(* IEC 61131-3 sources: Lasal/CPU_5344_V01/Class/Bit2ByteConversion_outputs, 1 file *)

(* ---- Bit2ByteConversion_outputs.st ---- *)
(*!
<Class
	Name               = "Bit2ByteConversion_outputs"
	Revision           = "0.1"
	RealtimeTask       = "false"
	CyclicTask         = "false"
	BackgroundTask     = "false"
	Sigmatek           = "false"
	OSInterface        = "false"
	HighPriority       = "false"
	Automatic          = "false"
	UpdateMode         = "Prescan"
	SharedCommandTable = "true"
	Objectsize         = "(390,2040)">
	<Channels>
		<Server Name="Bit1" Visualized="true" Initialize="false" WriteProtected="false" Retentive="false"/>
		<Server Name="Bit10" Visualized="true" Initialize="false" WriteProtected="false" Retentive="false"/>
		<Server Name="Bit11" Visualized="true" Initialize="false" WriteProtected="false" Retentive="false"/>
		<Server Name="Bit12" Visualized="true" Initialize="false" WriteProtected="false" Retentive="false"/>
		<Server Name="Bit13" Visualized="true" Initialize="false" WriteProtected="false" Retentive="false"/>
		<Server Name="Bit14" Visualized="true" Initialize="false" WriteProtected="false" Retentive="false"/>
		<Server Name="Bit15" Visualized="true" Initialize="false" WriteProtected="false" Retentive="false"/>
		<Server Name="Bit16" Visualized="true" Initialize="false" WriteProtected="false" Retentive="false"/>
		<Server Name="Bit17" Visualized="true" Initialize="false" WriteProtected="false" Retentive="false"/>
		<Server Name="Bit18" Visualized="true" Initialize="false" WriteProtected="false" Retentive="false"/>
		<Server Name="Bit19" Visualized="true" Initialize="false" WriteProtected="false" Retentive="false"/>
		<Server Name="Bit2" Visualized="true" Initialize="false" WriteProtected="false" Retentive="false"/>
		<Server Name="Bit20" Visualized="true" Initialize="false" WriteProtected="false" Retentive="false"/>
		<Server Name="Bit21" Visualized="true" Initialize="false" WriteProtected="false" Retentive="false"/>
		<Server Name="Bit22" Visualized="true" Initialize="false" WriteProtected="false" Retentive="false"/>
		<Server Name="Bit23" Visualized="true" Initialize="false" WriteProtected="false" Retentive="false"/>
		<Server Name="Bit24" Visualized="true" Initialize="false" WriteProtected="false" Retentive="false"/>
		<Server Name="Bit25" Visualized="true" Initialize="false" WriteProtected="false" Retentive="false"/>
		<Server Name="Bit26" Visualized="true" Initialize="false" WriteProtected="false" Retentive="false"/>
		<Server Name="Bit27" Visualized="true" Initialize="false" WriteProtected="false" Retentive="false"/>
		<Server Name="Bit28" Visualized="true" Initialize="false" WriteProtected="false" Retentive="false"/>
		<Server Name="Bit29" Visualized="true" Initialize="false" WriteProtected="false" Retentive="false"/>
		<Server Name="Bit3" Visualized="true" Initialize="false" WriteProtected="false" Retentive="false"/>
		<Server Name="Bit30" Visualized="true" Initialize="false" WriteProtected="false" Retentive="false"/>
		<Server Name="Bit31" Visualized="true" Initialize="false" WriteProtected="false" Retentive="false"/>
		<Server Name="Bit32" Visualized="true" Initialize="false" WriteProtected="false" Retentive="false"/>
		<Server Name="Bit4" Visualized="true" Initialize="false" WriteProtected="false" Retentive="false"/>
		<Server Name="Bit5" Visualized="true" Initialize="false" WriteProtected="false" Retentive="false"/>
		<Server Name="Bit6" Visualized="true" Initialize="false" WriteProtected="false" Retentive="false"/>
		<Server Name="Bit7" Visualized="true" Initialize="false" WriteProtected="false" Retentive="false"/>
		<Server Name="Bit8" Visualized="true" Initialize="false" WriteProtected="false" Retentive="false"/>
		<Server Name="Bit9" Visualized="true" Initialize="false" WriteProtected="false" Retentive="false"/>
		<Server Name="BitValue" Visualized="false" Initialize="false" WriteProtected="true" Retentive="false"/>
		<Client Name="BValue" Required="false" Internal="false"/>
	</Channels>
	<RevDoku>
		<Owner Company="Intecon" Author="Richard Fierkens"/>
		<Dokumentation Revision="0.1" Date="2011-12-28" Author="Richard Fierkens" Company="Intecon" Description="Write timedelay is removed.&#13;&#10;Read timedelay is set to 10mSec."/>
		<Dokumentation Revision="0.0" Date="2011-12-27" Author="Johan Embregts" Company="SigmaControl" Description="Created."/>
	</RevDoku>
</Class>
*)
Bit2ByteConversion_outputs : CLASS
  //Servers:
	BitValue 	: SvrChCmd_BDINT;
	Bit1 	: SvrCh_DINT;
	Bit2 	: SvrCh_DINT;
	Bit3 	: SvrCh_DINT;
	Bit4 	: SvrCh_DINT;
	Bit5 	: SvrCh_DINT;
	Bit6 	: SvrCh_DINT;
	Bit7 	: SvrCh_DINT;
	Bit8 	: SvrCh_DINT;
	Bit9 	: SvrCh_DINT;
	Bit10 	: SvrCh_DINT;
	Bit11 	: SvrCh_DINT;
	Bit12 	: SvrCh_DINT;
	Bit13 	: SvrCh_DINT;
	Bit14 	: SvrCh_DINT;
	Bit15 	: SvrCh_DINT;
	Bit16 	: SvrCh_DINT;
	Bit17 	: SvrCh_DINT;
	Bit18 	: SvrCh_DINT;
	Bit19 	: SvrCh_DINT;
	Bit20 	: SvrCh_DINT;
	Bit21 	: SvrCh_DINT;
	Bit22 	: SvrCh_DINT;
	Bit23 	: SvrCh_DINT;
	Bit24 	: SvrCh_DINT;
	Bit25 	: SvrCh_DINT;
	Bit26 	: SvrCh_DINT;
	Bit27 	: SvrCh_DINT;
	Bit28 	: SvrCh_DINT;
	Bit29 	: SvrCh_DINT;
	Bit30 	: SvrCh_DINT;
	Bit31 	: SvrCh_DINT;
	Bit32 	: SvrCh_DINT;
  //Clients:
	BValue 	: CltCh_BDINT;
  //Variables:
		tMark 	: UDINT;
  //Functions:

	FUNCTION VIRTUAL ReadMe;

	FUNCTION VIRTUAL WriteMe;

	FUNCTION VIRTUAL GLOBAL Bit1::Read
		VAR_OUTPUT
			output (EAX) 	: DINT;
		END_VAR;

	FUNCTION VIRTUAL GLOBAL Bit1::Write
		VAR_INPUT
			input (EAX) 	: DINT;
		END_VAR
		VAR_OUTPUT
			result (EAX) 	: DINT;
		END_VAR;

	FUNCTION VIRTUAL GLOBAL Bit2::Read
		VAR_OUTPUT
			output (EAX) 	: DINT;
		END_VAR;

	FUNCTION VIRTUAL GLOBAL Bit2::Write
		VAR_INPUT
			input (EAX) 	: DINT;
		END_VAR
		VAR_OUTPUT
			result (EAX) 	: DINT;
		END_VAR;

	FUNCTION VIRTUAL GLOBAL Bit3::Read
		VAR_OUTPUT
			output (EAX) 	: DINT;
		END_VAR;

	FUNCTION VIRTUAL GLOBAL Bit3::Write
		VAR_INPUT
			input (EAX) 	: DINT;
		END_VAR
		VAR_OUTPUT
			result (EAX) 	: DINT;
		END_VAR;

	FUNCTION VIRTUAL GLOBAL Bit4::Read
		VAR_OUTPUT
			output (EAX) 	: DINT;
		END_VAR;

	FUNCTION VIRTUAL GLOBAL Bit4::Write
		VAR_INPUT
			input (EAX) 	: DINT;
		END_VAR
		VAR_OUTPUT
			result (EAX) 	: DINT;
		END_VAR;

	FUNCTION VIRTUAL GLOBAL Bit5::Read
		VAR_OUTPUT
			output (EAX) 	: DINT;
		END_VAR;

	FUNCTION VIRTUAL GLOBAL Bit5::Write
		VAR_INPUT
			input (EAX) 	: DINT;
		END_VAR
		VAR_OUTPUT
			result (EAX) 	: DINT;
		END_VAR;

	FUNCTION VIRTUAL GLOBAL Bit6::Read
		VAR_OUTPUT
			output (EAX) 	: DINT;
		END_VAR;

	FUNCTION VIRTUAL GLOBAL Bit6::Write
		VAR_INPUT
			input (EAX) 	: DINT;
		END_VAR
		VAR_OUTPUT
			result (EAX) 	: DINT;
		END_VAR;

	FUNCTION VIRTUAL GLOBAL Bit7::Read
		VAR_OUTPUT
			output (EAX) 	: DINT;
		END_VAR;

	FUNCTION VIRTUAL GLOBAL Bit7::Write
		VAR_INPUT
			input (EAX) 	: DINT;
		END_VAR
		VAR_OUTPUT
			result (EAX) 	: DINT;
		END_VAR;

	FUNCTION VIRTUAL GLOBAL Bit8::Read
		VAR_OUTPUT
			output (EAX) 	: DINT;
		END_VAR;

	FUNCTION VIRTUAL GLOBAL Bit8::Write
		VAR_INPUT
			input (EAX) 	: DINT;
		END_VAR
		VAR_OUTPUT
			result (EAX) 	: DINT;
		END_VAR;

	FUNCTION VIRTUAL GLOBAL Bit9::Read
		VAR_OUTPUT
			output (EAX) 	: DINT;
		END_VAR;

	FUNCTION VIRTUAL GLOBAL Bit9::Write
		VAR_INPUT
			input (EAX) 	: DINT;
		END_VAR
		VAR_OUTPUT
			result (EAX) 	: DINT;
		END_VAR;

	FUNCTION VIRTUAL GLOBAL Bit10::Read
		VAR_OUTPUT
			output (EAX) 	: DINT;
		END_VAR;

	FUNCTION VIRTUAL GLOBAL Bit10::Write
		VAR_INPUT
			input (EAX) 	: DINT;
		END_VAR
		VAR_OUTPUT
			result (EAX) 	: DINT;
		END_VAR;

	FUNCTION VIRTUAL GLOBAL Bit11::Read
		VAR_OUTPUT
			output (EAX) 	: DINT;
		END_VAR;

	FUNCTION VIRTUAL GLOBAL Bit11::Write
		VAR_INPUT
			input (EAX) 	: DINT;
		END_VAR
		VAR_OUTPUT
			result (EAX) 	: DINT;
		END_VAR;

	FUNCTION VIRTUAL GLOBAL Bit12::Read
		VAR_OUTPUT
			output (EAX) 	: DINT;
		END_VAR;

	FUNCTION VIRTUAL GLOBAL Bit12::Write
		VAR_INPUT
			input (EAX) 	: DINT;
		END_VAR
		VAR_OUTPUT
			result (EAX) 	: DINT;
		END_VAR;

	FUNCTION VIRTUAL GLOBAL Bit13::Read
		VAR_OUTPUT
			output (EAX) 	: DINT;
		END_VAR;

	FUNCTION VIRTUAL GLOBAL Bit13::Write
		VAR_INPUT
			input (EAX) 	: DINT;
		END_VAR
		VAR_OUTPUT
			result (EAX) 	: DINT;
		END_VAR;

	FUNCTION VIRTUAL GLOBAL Bit14::Read
		VAR_OUTPUT
			output (EAX) 	: DINT;
		END_VAR;

	FUNCTION VIRTUAL GLOBAL Bit14::Write
		VAR_INPUT
			input (EAX) 	: DINT;
		END_VAR
		VAR_OUTPUT
			result (EAX) 	: DINT;
		END_VAR;

	FUNCTION VIRTUAL GLOBAL Bit15::Read
		VAR_OUTPUT
			output (EAX) 	: DINT;
		END_VAR;

	FUNCTION VIRTUAL GLOBAL Bit15::Write
		VAR_INPUT
			input (EAX) 	: DINT;
		END_VAR
		VAR_OUTPUT
			result (EAX) 	: DINT;
		END_VAR;

	FUNCTION VIRTUAL GLOBAL Bit16::Read
		VAR_OUTPUT
			output (EAX) 	: DINT;
		END_VAR;

	FUNCTION VIRTUAL GLOBAL Bit16::Write
		VAR_INPUT
			input (EAX) 	: DINT;
		END_VAR
		VAR_OUTPUT
			result (EAX) 	: DINT;
		END_VAR;

	FUNCTION VIRTUAL GLOBAL Bit17::Read
		VAR_OUTPUT
			output (EAX) 	: DINT;
		END_VAR;

	FUNCTION VIRTUAL GLOBAL Bit17::Write
		VAR_INPUT
			input (EAX) 	: DINT;
		END_VAR
		VAR_OUTPUT
			result (EAX) 	: DINT;
		END_VAR;

	FUNCTION VIRTUAL GLOBAL Bit18::Read
		VAR_OUTPUT
			output (EAX) 	: DINT;
		END_VAR;

	FUNCTION VIRTUAL GLOBAL Bit18::Write
		VAR_INPUT
			input (EAX) 	: DINT;
		END_VAR
		VAR_OUTPUT
			result (EAX) 	: DINT;
		END_VAR;

	FUNCTION VIRTUAL GLOBAL Bit19::Read
		VAR_OUTPUT
			output (EAX) 	: DINT;
		END_VAR;

	FUNCTION VIRTUAL GLOBAL Bit19::Write
		VAR_INPUT
			input (EAX) 	: DINT;
		END_VAR
		VAR_OUTPUT
			result (EAX) 	: DINT;
		END_VAR;

	FUNCTION VIRTUAL GLOBAL Bit20::Read
		VAR_OUTPUT
			output (EAX) 	: DINT;
		END_VAR;

	FUNCTION VIRTUAL GLOBAL Bit20::Write
		VAR_INPUT
			input (EAX) 	: DINT;
		END_VAR
		VAR_OUTPUT
			result (EAX) 	: DINT;
		END_VAR;

	FUNCTION VIRTUAL GLOBAL Bit21::Read
		VAR_OUTPUT
			output (EAX) 	: DINT;
		END_VAR;

	FUNCTION VIRTUAL GLOBAL Bit21::Write
		VAR_INPUT
			input (EAX) 	: DINT;
		END_VAR
		VAR_OUTPUT
			result (EAX) 	: DINT;
		END_VAR;

	FUNCTION VIRTUAL GLOBAL Bit22::Read
		VAR_OUTPUT
			output (EAX) 	: DINT;
		END_VAR;

	FUNCTION VIRTUAL GLOBAL Bit22::Write
		VAR_INPUT
			input (EAX) 	: DINT;
		END_VAR
		VAR_OUTPUT
			result (EAX) 	: DINT;
		END_VAR;

	FUNCTION VIRTUAL GLOBAL Bit23::Read
		VAR_OUTPUT
			output (EAX) 	: DINT;
		END_VAR;

	FUNCTION VIRTUAL GLOBAL Bit23::Write
		VAR_INPUT
			input (EAX) 	: DINT;
		END_VAR
		VAR_OUTPUT
			result (EAX) 	: DINT;
		END_VAR;

	FUNCTION VIRTUAL GLOBAL Bit24::Read
		VAR_OUTPUT
			output (EAX) 	: DINT;
		END_VAR;

	FUNCTION VIRTUAL GLOBAL Bit24::Write
		VAR_INPUT
			input (EAX) 	: DINT;
		END_VAR
		VAR_OUTPUT
			result (EAX) 	: DINT;
		END_VAR;

	FUNCTION VIRTUAL GLOBAL Bit25::Read
		VAR_OUTPUT
			output (EAX) 	: DINT;
		END_VAR;

	FUNCTION VIRTUAL GLOBAL Bit25::Write
		VAR_INPUT
			input (EAX) 	: DINT;
		END_VAR
		VAR_OUTPUT
			result (EAX) 	: DINT;
		END_VAR;

	FUNCTION VIRTUAL GLOBAL Bit26::Read
		VAR_OUTPUT
			output (EAX) 	: DINT;
		END_VAR;

	FUNCTION VIRTUAL GLOBAL Bit26::Write
		VAR_INPUT
			input (EAX) 	: DINT;
		END_VAR
		VAR_OUTPUT
			result (EAX) 	: DINT;
		END_VAR;

	FUNCTION VIRTUAL GLOBAL Bit27::Read
		VAR_OUTPUT
			output (EAX) 	: DINT;
		END_VAR;

	FUNCTION VIRTUAL GLOBAL Bit27::Write
		VAR_INPUT
			input (EAX) 	: DINT;
		END_VAR
		VAR_OUTPUT
			result (EAX) 	: DINT;
		END_VAR;

	FUNCTION VIRTUAL GLOBAL Bit28::Read
		VAR_OUTPUT
			output (EAX) 	: DINT;
		END_VAR;

	FUNCTION VIRTUAL GLOBAL Bit28::Write
		VAR_INPUT
			input (EAX) 	: DINT;
		END_VAR
		VAR_OUTPUT
			result (EAX) 	: DINT;
		END_VAR;

	FUNCTION VIRTUAL GLOBAL Bit29::Read
		VAR_OUTPUT
			output (EAX) 	: DINT;
		END_VAR;

	FUNCTION VIRTUAL GLOBAL Bit29::Write
		VAR_INPUT
			input (EAX) 	: DINT;
		END_VAR
		VAR_OUTPUT
			result (EAX) 	: DINT;
		END_VAR;

	FUNCTION VIRTUAL GLOBAL Bit30::Read
		VAR_OUTPUT
			output (EAX) 	: DINT;
		END_VAR;

	FUNCTION VIRTUAL GLOBAL Bit30::Write
		VAR_INPUT
			input (EAX) 	: DINT;
		END_VAR
		VAR_OUTPUT
			result (EAX) 	: DINT;
		END_VAR;

	FUNCTION VIRTUAL GLOBAL Bit31::Read
		VAR_OUTPUT
			output (EAX) 	: DINT;
		END_VAR;

	FUNCTION VIRTUAL GLOBAL Bit31::Write
		VAR_INPUT
			input (EAX) 	: DINT;
		END_VAR
		VAR_OUTPUT
			result (EAX) 	: DINT;
		END_VAR;

	FUNCTION VIRTUAL GLOBAL Bit32::Read
		VAR_OUTPUT
			output (EAX) 	: DINT;
		END_VAR;

	FUNCTION VIRTUAL GLOBAL Bit32::Write
		VAR_INPUT
			input (EAX) 	: DINT;
		END_VAR
		VAR_OUTPUT
			result (EAX) 	: DINT;
		END_VAR;
  //Tables:
	FUNCTION @STD
		VAR_OUTPUT
			ret_code	: CONFSTATES;
		END_VAR;
	FUNCTION GLOBAL TAB @CT_;
END_CLASS;

#define cMaxUpdateTime  10 // mSec

FUNCTION VIRTUAL GLOBAL Bit2ByteConversion_outputs::Bit1::Read
	VAR_OUTPUT
		output (EAX) 	: DINT;
	END_VAR

  ReadMe();
	output := Bit1;

END_FUNCTION

FUNCTION VIRTUAL GLOBAL Bit2ByteConversion_outputs::Bit2::Read
	VAR_OUTPUT
		output (EAX) 	: DINT;
	END_VAR

  ReadMe();
	output := Bit2;

END_FUNCTION

FUNCTION VIRTUAL GLOBAL Bit2ByteConversion_outputs::Bit3::Read
	VAR_OUTPUT
		output (EAX) 	: DINT;
	END_VAR

  ReadMe();
	output := Bit3;

END_FUNCTION

FUNCTION VIRTUAL GLOBAL Bit2ByteConversion_outputs::Bit4::Read
	VAR_OUTPUT
		output (EAX) 	: DINT;
	END_VAR

  ReadMe();
	output := Bit4;

END_FUNCTION

FUNCTION VIRTUAL GLOBAL Bit2ByteConversion_outputs::Bit5::Read
	VAR_OUTPUT
		output (EAX) 	: DINT;
	END_VAR

  ReadMe();
	output := Bit5;

END_FUNCTION

FUNCTION VIRTUAL GLOBAL Bit2ByteConversion_outputs::Bit6::Read
	VAR_OUTPUT
		output (EAX) 	: DINT;
	END_VAR

  ReadMe();
	output := Bit6;

END_FUNCTION

FUNCTION VIRTUAL GLOBAL Bit2ByteConversion_outputs::Bit7::Read
	VAR_OUTPUT
		output (EAX) 	: DINT;
	END_VAR

  ReadMe();
	output := Bit7;

END_FUNCTION

FUNCTION VIRTUAL GLOBAL Bit2ByteConversion_outputs::Bit8::Read
	VAR_OUTPUT
		output (EAX) 	: DINT;
	END_VAR

  ReadMe();
	output := Bit8;

END_FUNCTION

FUNCTION VIRTUAL GLOBAL Bit2ByteConversion_outputs::Bit9::Read
	VAR_OUTPUT
		output (EAX) 	: DINT;
	END_VAR

  ReadMe();
	output := Bit9;

END_FUNCTION

FUNCTION VIRTUAL GLOBAL Bit2ByteConversion_outputs::Bit10::Read
	VAR_OUTPUT
		output (EAX) 	: DINT;
	END_VAR

  ReadMe();
	output := Bit10;

END_FUNCTION

FUNCTION VIRTUAL GLOBAL Bit2ByteConversion_outputs::Bit11::Read
	VAR_OUTPUT
		output (EAX) 	: DINT;
	END_VAR

  ReadMe();
	output := Bit11;

END_FUNCTION

FUNCTION VIRTUAL GLOBAL Bit2ByteConversion_outputs::Bit12::Read
	VAR_OUTPUT
		output (EAX) 	: DINT;
	END_VAR

  ReadMe();
	output := Bit12;

END_FUNCTION

FUNCTION VIRTUAL GLOBAL Bit2ByteConversion_outputs::Bit13::Read
	VAR_OUTPUT
		output (EAX) 	: DINT;
	END_VAR

  ReadMe();
	output := Bit13;

END_FUNCTION

FUNCTION VIRTUAL GLOBAL Bit2ByteConversion_outputs::Bit14::Read
	VAR_OUTPUT
		output (EAX) 	: DINT;
	END_VAR

  ReadMe();
	output := Bit14;

END_FUNCTION

FUNCTION VIRTUAL GLOBAL Bit2ByteConversion_outputs::Bit15::Read
	VAR_OUTPUT
		output (EAX) 	: DINT;
	END_VAR

  ReadMe();
	output := Bit15;

END_FUNCTION

FUNCTION VIRTUAL GLOBAL Bit2ByteConversion_outputs::Bit16::Read
	VAR_OUTPUT
		output (EAX) 	: DINT;
	END_VAR

  ReadMe();
	output := Bit16;

END_FUNCTION

FUNCTION VIRTUAL GLOBAL Bit2ByteConversion_outputs::Bit17::Read
	VAR_OUTPUT
		output (EAX) 	: DINT;
	END_VAR

  ReadMe();
	output := Bit17;

END_FUNCTION

FUNCTION VIRTUAL GLOBAL Bit2ByteConversion_outputs::Bit18::Read
	VAR_OUTPUT
		output (EAX) 	: DINT;
	END_VAR

  ReadMe();
	output := Bit18;

END_FUNCTION

FUNCTION VIRTUAL GLOBAL Bit2ByteConversion_outputs::Bit19::Read
	VAR_OUTPUT
		output (EAX) 	: DINT;
	END_VAR

  ReadMe();
	output := Bit19;

END_FUNCTION

FUNCTION VIRTUAL GLOBAL Bit2ByteConversion_outputs::Bit20::Read
	VAR_OUTPUT
		output (EAX) 	: DINT;
	END_VAR

  ReadMe();
	output := Bit20;

END_FUNCTION

FUNCTION VIRTUAL GLOBAL Bit2ByteConversion_outputs::Bit21::Read
	VAR_OUTPUT
		output (EAX) 	: DINT;
	END_VAR

  ReadMe();
	output := Bit21;

END_FUNCTION

FUNCTION VIRTUAL GLOBAL Bit2ByteConversion_outputs::Bit22::Read
	VAR_OUTPUT
		output (EAX) 	: DINT;
	END_VAR

  ReadMe();
	output := Bit22;

END_FUNCTION

FUNCTION VIRTUAL GLOBAL Bit2ByteConversion_outputs::Bit23::Read
	VAR_OUTPUT
		output (EAX) 	: DINT;
	END_VAR

  ReadMe();
	output := Bit23;

END_FUNCTION

FUNCTION VIRTUAL GLOBAL Bit2ByteConversion_outputs::Bit24::Read
	VAR_OUTPUT
		output (EAX) 	: DINT;
	END_VAR

  ReadMe();
	output := Bit24;

END_FUNCTION

FUNCTION VIRTUAL GLOBAL Bit2ByteConversion_outputs::Bit25::Read
	VAR_OUTPUT
		output (EAX) 	: DINT;
	END_VAR

  ReadMe();
	output := Bit25;

END_FUNCTION

FUNCTION VIRTUAL GLOBAL Bit2ByteConversion_outputs::Bit26::Read
	VAR_OUTPUT
		output (EAX) 	: DINT;
	END_VAR

  ReadMe();
	output := Bit26;

END_FUNCTION

FUNCTION VIRTUAL GLOBAL Bit2ByteConversion_outputs::Bit27::Read
	VAR_OUTPUT
		output (EAX) 	: DINT;
	END_VAR

  ReadMe();
	output := Bit27;

END_FUNCTION

FUNCTION VIRTUAL GLOBAL Bit2ByteConversion_outputs::Bit28::Read
	VAR_OUTPUT
		output (EAX) 	: DINT;
	END_VAR

  ReadMe();
	output := Bit28;

END_FUNCTION

FUNCTION VIRTUAL GLOBAL Bit2ByteConversion_outputs::Bit29::Read
	VAR_OUTPUT
		output (EAX) 	: DINT;
	END_VAR

  ReadMe();
	output := Bit29;

END_FUNCTION

FUNCTION VIRTUAL GLOBAL Bit2ByteConversion_outputs::Bit30::Read
	VAR_OUTPUT
		output (EAX) 	: DINT;
	END_VAR

  ReadMe();
	output := Bit30;

END_FUNCTION

FUNCTION VIRTUAL GLOBAL Bit2ByteConversion_outputs::Bit31::Read
	VAR_OUTPUT
		output (EAX) 	: DINT;
	END_VAR

  ReadMe();
	output := Bit31;

END_FUNCTION

FUNCTION VIRTUAL GLOBAL Bit2ByteConversion_outputs::Bit32::Read
	VAR_OUTPUT
		output (EAX) 	: DINT;
	END_VAR

  ReadMe();
	output := Bit32;

END_FUNCTION

FUNCTION VIRTUAL GLOBAL Bit2ByteConversion_outputs::Bit1::Write
	VAR_INPUT
		input (EAX) 	: DINT;
	END_VAR
	VAR_OUTPUT
		result (EAX) 	: DINT;
	END_VAR

  Bit1 := input and 2#1;
	BValue.1 := to_Bool( Bit1);
  WriteMe();
 	result := Bit1;

END_FUNCTION

FUNCTION VIRTUAL GLOBAL Bit2ByteConversion_outputs::Bit2::Write
	VAR_INPUT
		input (EAX) 	: DINT;
	END_VAR
	VAR_OUTPUT
		result (EAX) 	: DINT;
	END_VAR

  Bit2 := input and 2#1;
	BValue.2 := to_Bool( Bit2);
  WriteMe();
 	result := Bit2;

END_FUNCTION

FUNCTION VIRTUAL GLOBAL Bit2ByteConversion_outputs::Bit3::Write
	VAR_INPUT
		input (EAX) 	: DINT;
	END_VAR
	VAR_OUTPUT
		result (EAX) 	: DINT;
	END_VAR

  Bit3 := input and 2#1;
	BValue.3 := to_Bool( Bit3);
  WriteMe();
 	result := Bit3;

END_FUNCTION

FUNCTION VIRTUAL GLOBAL Bit2ByteConversion_outputs::Bit4::Write
	VAR_INPUT
		input (EAX) 	: DINT;
	END_VAR
	VAR_OUTPUT
		result (EAX) 	: DINT;
	END_VAR

  Bit4 := input and 2#1;
	BValue.4 := to_Bool( Bit4);
  WriteMe();
 	result := Bit4;

END_FUNCTION

FUNCTION VIRTUAL GLOBAL Bit2ByteConversion_outputs::Bit5::Write
	VAR_INPUT
		input (EAX) 	: DINT;
	END_VAR
	VAR_OUTPUT
		result (EAX) 	: DINT;
	END_VAR

  Bit5 := input and 2#1;
	BValue.5 := to_Bool( Bit5);
  WriteMe();
 	result := Bit5;

END_FUNCTION

FUNCTION VIRTUAL GLOBAL Bit2ByteConversion_outputs::Bit6::Write
	VAR_INPUT
		input (EAX) 	: DINT;
	END_VAR
	VAR_OUTPUT
		result (EAX) 	: DINT;
	END_VAR

  Bit6 := input and 2#1;
	BValue.6 := to_Bool( Bit6);
  WriteMe();
 	result := Bit6;

END_FUNCTION

FUNCTION VIRTUAL GLOBAL Bit2ByteConversion_outputs::Bit7::Write
	VAR_INPUT
		input (EAX) 	: DINT;
	END_VAR
	VAR_OUTPUT
		result (EAX) 	: DINT;
	END_VAR

  Bit7 := input and 2#1;
	BValue.7 := to_Bool( Bit7);
  WriteMe();
 	result := Bit7;

END_FUNCTION

FUNCTION VIRTUAL GLOBAL Bit2ByteConversion_outputs::Bit8::Write
	VAR_INPUT
		input (EAX) 	: DINT;
	END_VAR
	VAR_OUTPUT
		result (EAX) 	: DINT;
	END_VAR

  Bit8 := input and 2#1;
	BValue.8 := to_Bool( Bit8);
  WriteMe();
 	result := Bit8;

END_FUNCTION

FUNCTION VIRTUAL GLOBAL Bit2ByteConversion_outputs::Bit9::Write
	VAR_INPUT
		input (EAX) 	: DINT;
	END_VAR
	VAR_OUTPUT
		result (EAX) 	: DINT;
	END_VAR

  Bit9 := input and 2#1;
	BValue.9 := to_Bool( Bit9);
  WriteMe();
 	result := Bit9;

END_FUNCTION

FUNCTION VIRTUAL GLOBAL Bit2ByteConversion_outputs::Bit10::Write
	VAR_INPUT
		input (EAX) 	: DINT;
	END_VAR
	VAR_OUTPUT
		result (EAX) 	: DINT;
	END_VAR

  Bit10 := input and 2#1;
	BValue.10 := to_Bool( Bit10);
  WriteMe();
 	result := Bit10;

END_FUNCTION

FUNCTION VIRTUAL GLOBAL Bit2ByteConversion_outputs::Bit11::Write
	VAR_INPUT
		input (EAX) 	: DINT;
	END_VAR
	VAR_OUTPUT
		result (EAX) 	: DINT;
	END_VAR

  Bit11 := input and 2#1;
	BValue.11 := to_Bool( Bit11);
  WriteMe();
 	result := Bit11;

END_FUNCTION

FUNCTION VIRTUAL GLOBAL Bit2ByteConversion_outputs::Bit12::Write
	VAR_INPUT
		input (EAX) 	: DINT;
	END_VAR
	VAR_OUTPUT
		result (EAX) 	: DINT;
	END_VAR

  Bit12 := input and 2#1;
	BValue.12 := to_Bool( Bit12);
  WriteMe();
 	result := Bit12;

END_FUNCTION

FUNCTION VIRTUAL GLOBAL Bit2ByteConversion_outputs::Bit13::Write
	VAR_INPUT
		input (EAX) 	: DINT;
	END_VAR
	VAR_OUTPUT
		result (EAX) 	: DINT;
	END_VAR

  Bit13 := input and 2#1;
	BValue.13 := to_Bool( Bit13);
  WriteMe();
 	result := Bit13;

END_FUNCTION

FUNCTION VIRTUAL GLOBAL Bit2ByteConversion_outputs::Bit14::Write
	VAR_INPUT
		input (EAX) 	: DINT;
	END_VAR
	VAR_OUTPUT
		result (EAX) 	: DINT;
	END_VAR

  Bit14 := input and 2#1;
	BValue.14 := to_Bool( Bit14);
  WriteMe();
 	result := Bit14;

END_FUNCTION

FUNCTION VIRTUAL GLOBAL Bit2ByteConversion_outputs::Bit15::Write
	VAR_INPUT
		input (EAX) 	: DINT;
	END_VAR
	VAR_OUTPUT
		result (EAX) 	: DINT;
	END_VAR

  Bit15 := input and 2#1;
	BValue.15 := to_Bool( Bit15);
  WriteMe();
 	result := Bit15;

END_FUNCTION

FUNCTION VIRTUAL GLOBAL Bit2ByteConversion_outputs::Bit16::Write
	VAR_INPUT
		input (EAX) 	: DINT;
	END_VAR
	VAR_OUTPUT
		result (EAX) 	: DINT;
	END_VAR

  Bit16 := input and 2#1;
	BValue.16 := to_Bool( Bit16);
  WriteMe();
 	result := Bit16;

END_FUNCTION

FUNCTION VIRTUAL GLOBAL Bit2ByteConversion_outputs::Bit17::Write
	VAR_INPUT
		input (EAX) 	: DINT;
	END_VAR
	VAR_OUTPUT
		result (EAX) 	: DINT;
	END_VAR

  Bit17 := input and 2#1;
	BValue.17 := to_Bool( Bit17);
  WriteMe();
 	result := Bit17;

END_FUNCTION

FUNCTION VIRTUAL GLOBAL Bit2ByteConversion_outputs::Bit18::Write
	VAR_INPUT
		input (EAX) 	: DINT;
	END_VAR
	VAR_OUTPUT
		result (EAX) 	: DINT;
	END_VAR

  Bit18 := input and 2#1;
	BValue.18 := to_Bool( Bit18);
  WriteMe();
 	result := Bit18;

END_FUNCTION

FUNCTION VIRTUAL GLOBAL Bit2ByteConversion_outputs::Bit19::Write
	VAR_INPUT
		input (EAX) 	: DINT;
	END_VAR
	VAR_OUTPUT
		result (EAX) 	: DINT;
	END_VAR

  Bit19 := input and 2#1;
	BValue.19 := to_Bool( Bit19);
  WriteMe();
 	result := Bit19;

END_FUNCTION

FUNCTION VIRTUAL GLOBAL Bit2ByteConversion_outputs::Bit20::Write
	VAR_INPUT
		input (EAX) 	: DINT;
	END_VAR
	VAR_OUTPUT
		result (EAX) 	: DINT;
	END_VAR

  Bit20 := input and 2#1;
	BValue.20 := to_Bool( Bit20);
  WriteMe();
 	result := Bit20;

END_FUNCTION

FUNCTION VIRTUAL GLOBAL Bit2ByteConversion_outputs::Bit21::Write
	VAR_INPUT
		input (EAX) 	: DINT;
	END_VAR
	VAR_OUTPUT
		result (EAX) 	: DINT;
	END_VAR

  Bit21 := input and 2#1;
	BValue.21 := to_Bool( Bit21);
  WriteMe();
 	result := Bit21;

END_FUNCTION

FUNCTION VIRTUAL GLOBAL Bit2ByteConversion_outputs::Bit22::Write
	VAR_INPUT
		input (EAX) 	: DINT;
	END_VAR
	VAR_OUTPUT
		result (EAX) 	: DINT;
	END_VAR

  Bit22 := input and 2#1;
	BValue.22 := to_Bool( Bit22);
  WriteMe();
 	result := Bit22;

END_FUNCTION

FUNCTION VIRTUAL GLOBAL Bit2ByteConversion_outputs::Bit23::Write
	VAR_INPUT
		input (EAX) 	: DINT;
	END_VAR
	VAR_OUTPUT
		result (EAX) 	: DINT;
	END_VAR

  Bit23 := input and 2#1;
	BValue.23 := to_Bool( Bit23);
  WriteMe();
 	result := Bit23;

END_FUNCTION

FUNCTION VIRTUAL GLOBAL Bit2ByteConversion_outputs::Bit24::Write
	VAR_INPUT
		input (EAX) 	: DINT;
	END_VAR
	VAR_OUTPUT
		result (EAX) 	: DINT;
	END_VAR

  Bit24 := input and 2#1;
	BValue.24 := to_Bool( Bit24);
  WriteMe();
 	result := Bit24;

END_FUNCTION

FUNCTION VIRTUAL GLOBAL Bit2ByteConversion_outputs::Bit25::Write
	VAR_INPUT
		input (EAX) 	: DINT;
	END_VAR
	VAR_OUTPUT
		result (EAX) 	: DINT;
	END_VAR

  Bit25 := input and 2#1;
	BValue.25 := to_Bool( Bit25);
  WriteMe();
 	result := Bit25;

END_FUNCTION

FUNCTION VIRTUAL GLOBAL Bit2ByteConversion_outputs::Bit26::Write
	VAR_INPUT
		input (EAX) 	: DINT;
	END_VAR
	VAR_OUTPUT
		result (EAX) 	: DINT;
	END_VAR

  Bit26 := input and 2#1;
	BValue.26 := to_Bool( Bit26);
  WriteMe();
 	result := Bit26;

END_FUNCTION

FUNCTION VIRTUAL GLOBAL Bit2ByteConversion_outputs::Bit27::Write
	VAR_INPUT
		input (EAX) 	: DINT;
	END_VAR
	VAR_OUTPUT
		result (EAX) 	: DINT;
	END_VAR

  Bit27 := input and 2#1;
	BValue.27 := to_Bool( Bit27);
  WriteMe();
 	result := Bit27;

END_FUNCTION

FUNCTION VIRTUAL GLOBAL Bit2ByteConversion_outputs::Bit28::Write
	VAR_INPUT
		input (EAX) 	: DINT;
	END_VAR
	VAR_OUTPUT
		result (EAX) 	: DINT;
	END_VAR

  Bit28 := input and 2#1;
	BValue.28 := to_Bool( Bit28);
  WriteMe();
 	result := Bit28;

END_FUNCTION

FUNCTION VIRTUAL GLOBAL Bit2ByteConversion_outputs::Bit29::Write
	VAR_INPUT
		input (EAX) 	: DINT;
	END_VAR
	VAR_OUTPUT
		result (EAX) 	: DINT;
	END_VAR

  Bit29 := input and 2#1;
	BValue.29 := to_Bool( Bit29);
  WriteMe();
 	result := Bit29;

END_FUNCTION

FUNCTION VIRTUAL GLOBAL Bit2ByteConversion_outputs::Bit30::Write
	VAR_INPUT
		input (EAX) 	: DINT;
	END_VAR
	VAR_OUTPUT
		result (EAX) 	: DINT;
	END_VAR

  Bit30 := input and 2#1;
	BValue.30 := to_Bool( Bit30);
  WriteMe();
 	result := Bit30;

END_FUNCTION

FUNCTION VIRTUAL GLOBAL Bit2ByteConversion_outputs::Bit31::Write
	VAR_INPUT
		input (EAX) 	: DINT;
	END_VAR
	VAR_OUTPUT
		result (EAX) 	: DINT;
	END_VAR

  Bit31 := input and 2#1;
	BValue.31 := to_Bool( Bit31);
  WriteMe();
 	result := Bit31;

END_FUNCTION

FUNCTION VIRTUAL GLOBAL Bit2ByteConversion_outputs::Bit32::Write
	VAR_INPUT
		input (EAX) 	: DINT;
	END_VAR
	VAR_OUTPUT
		result (EAX) 	: DINT;
	END_VAR

  Bit32 := input and 2#1;
	BValue.32 := to_Bool( Bit32);
  WriteMe();
 	result := Bit32;

END_FUNCTION

FUNCTION VIRTUAL Bit2ByteConversion_outputs::ReadMe

  if ops.tAbsolute- tMark> cMaxUpdateTime then
    BitValue  := BValue := BValue.Read();
    Bit1  := BValue.1;
    Bit2  := BValue.2;
    Bit3  := BValue.3;
    Bit4  := BValue.4;
    Bit5  := BValue.5;
    Bit6  := BValue.6;
    Bit7  := BValue.7;
    Bit8  := BValue.8;
    Bit9  := BValue.9;
    Bit10 := BValue.10;
    Bit11 := BValue.11;
    Bit12 := BValue.12;
    Bit13 := BValue.13;
    Bit14 := BValue.14;
    Bit15 := BValue.15;
    Bit16 := BValue.16;
    Bit17 := BValue.17;
    Bit18 := BValue.18;
    Bit19 := BValue.19;
    Bit20 := BValue.20;
    Bit21 := BValue.21;
    Bit22 := BValue.22;
    Bit23 := BValue.23;
    Bit24 := BValue.24;
    Bit25 := BValue.25;
    Bit26 := BValue.26;
    Bit27 := BValue.27;
    Bit28 := BValue.28;
    Bit29 := BValue.29;
    Bit30 := BValue.30;
    Bit31 := BValue.31;
    Bit32 := BValue.32;
    tMark := ops.tAbsolute;
  end_if;

END_FUNCTION

FUNCTION VIRTUAL Bit2ByteConversion_outputs::WriteMe

 // if ops.tAbsolute- tMark> cMaxUpdateTime then
    BitValue  := to_Udint( BValue.Write( BValue));
    tMark := ops.tAbsolute;
 // end_if;

END_FUNCTION
